FUNCTION F_TrimRightSpace : STRING
VAR_INPUT
	 strIn : STRING;
END_VAR
VAR
	  nLen : INT;
END_VAR

F_TrimRightSpace := strIn;

	nLen := LEN(F_TrimRightSpace);
	
	WHILE (nLen > 0) AND MID(F_TrimRightSpace,1,nLen)=' ' DO
		nLen := nLen - 1;
	END_WHILE
	F_TrimRightSpace := LEFT(F_TrimRightSpace, nLen);

END_FUNCTION

(* stored: Version 1.1.0.1, ProductVersion 3.1.4024.16
   POU F_TrimRightSpace: Id {16d7ff96-f89e-4e5a-8f9c-2ea2dac80d83}, SpecialFunc None *)
